// TIA Portal V20 export
TYPE "MotorVSDIOSet"
// stored: IsFailsafeCompliant false
   STRUCT
      InHand : Bool;
      AutoStartSignal : Bool;
      HandStartSignal : Bool;
      RunningFwdFB : Bool;
      RunningRevFB : Bool;
      VSDError : Bool;
      SystemHealthy : Bool;
      PreStartDone : Bool;
      InhibitMotor : Bool;
      FaultReset : Bool;
      FTTime : Real;
      EnableUPSTime : Real;
      FaultActive : Bool;
      Run : Bool;
      RunRev : Bool;
      UPSEnable : Bool;
      FTR : Bool;
      FTS : Bool;
      HrsRun : UDInt;
      Telemetry : Int;
      Alarm : Word;
      "Name" : String;
      HandIntervention : Bool;
      TryRunMotor : Bool;
      RecentStart : Bool;
      ShutdownComplete : Bool;
      ShutdownTime : Real;
      Shutdown : Bool;
      StopMotor : Bool;
      VSDWarning : Bool;
      HandSpeedInput : Real;
      AutoSpeedInput : Real;
      SpeedOutput : Int;
      SpeedPerc : Real;
      SpeedFB : Int;
      SpeedReached : Bool;
      AmpsFB : Real;
      OverTempFault : Bool;
      ThermalOLFault : Bool;
      TorqueLimitOk : Bool;
      VSDReady : Bool;
      VSDOpEnable : Bool;
      VSDOverSpeed : Bool;
      VSDUnderSpeed : Bool;
      RotationSensor : Bool;
      StartUpTime : Real;
      MaxRPM : Int;
   END_STRUCT;
END_TYPE
